TYPE ST_MachineControl :
STRUCT
	bPressureBeamLower : BOOL;
	bPressureBeamRaise : BOOL;
	bClamp : BOOL;
	bUnclamp: BOOL;
END_STRUCT
END_TYPE

(* stored: Version 1.1.0.1
   DUT ST_MachineControl: Id {daaa6b6a-c926-416c-a476-93c80d455284} *)
